PROGRAM MAIN
VAR
	record : ST_Record;
	bla : DWORD;
END_VAR

bla := record.test[9999];

END_PROGRAM

(* stored: Version 1.1.0.1, ProductVersion 3.1.4020.6
   POU MAIN: Id {282793d0-dd86-449b-919f-f07f679b0527}, SpecialFunc None *)
